TEXTLIST EventPriority
  2 = 'MiddleHigh'
  3 = 'Middle'
  4 = 'MiddleLow'
  5 = 'Low'
  255 = 'Unknown'
   = ''
END_TEXTLIST

(* stored: Version 1.1.0.1
   TextList EventPriority: Id {2110d44b-cf71-4202-a7df-49e677947f75} *)
